INTERFACE I_PersistentEventStorage

METHOD StoreEvent
VAR_INPUT
	stEvent:ST_Event;
END_VAR
END_METHOD

END_INTERFACE

(* stored: Version 1.1.0.1, ProductVersion 3.1.4024.12
   Itf I_PersistentEventStorage: Id {df0400e6-a321-497b-bf02-9f5070ca94eb}
   Method StoreEvent: Id {79462987-54b5-4f64-8125-f253a6f4e99e} *)
